ABB RobotStudio station: PROYECTO_PROGRAMACION_DE_ROBTOS.rsstnx

Station PROYECTO_PROGRAMACION_DE_ROBTOS (saved by RobotStudio 23.2.10395.0)
Controller IRB120_3_58_1, task T_ROB1: task frame (RAPID world) sits at (-1295.2, 4.92, 820) mm in the station
Controller IRB120_3_58, task T_ROB1: task frame (RAPID world) sits at (388.16, 1257.89, 820) mm in the station
Controller IRB120_3_58
  mechanical unit ROB_1: IRB120_3_58__01, 6 joints, base frame (0, -1249.97, 0) mm
Controller IRB120_3_58_1
  mechanical unit ROB_1: IRB120_3_58__01_2, 6 joints, base frame (0, 0, 0) mm
Layout (positions relative to the parent item):
  - IRB120_3_58__01 [mechanism, from %ABB.RobotStudio.Models.IRB120%\IRB120_3_58_G_01.rslib] at (388.16, 7.91, 820) mm; joint values [0, 0, 0, 0, 0.5236, 0] (rad or m)
  - CONVEYOR 1 [part, from %ABB.RobotStudio.Models.Conveyors%\Conveyor Guide 400.rslib] at (666.35, -202.61, 0) mm
  - CONVEYOR 2-1 [part, from %ABB.RobotStudio.Models.Conveyors%\Conveyor Guide 400.rslib] at (-1287.84, -701.07, 0) mm
  - CONVEYOR 2-2 [part, from %ABB.RobotStudio.Models.Conveyors%\Conveyor Guide 400.rslib] at (-1267.75, 333.06, 0) mm
  - CILINDRO_BASE 1 [part] at (385.3, 0, 0) mm, size 200 x 197 x 750 mm
  - BASE 1 [part] at (388.12, -2.42, 750) mm, size 300 x 298.4 x 70 mm
  - IRB120_3_58__01_2 [mechanism, from %ABB.RobotStudio.Models.IRB120%\IRB120_3_58_G_01.rslib] at (-1295.2, 4.92, 820) mm; joint values [0, 0, 0, 0, 0.5236, 0] (rad or m)
  - CILINDRO_BASE 2 [part] at (-1281.83, 0, 0) mm, size 200 x 197 x 750 mm
  - BASE 2 [part] at (-1282.88, 0.78, 750) mm, size 300 x 298.4 x 70 mm
